FUNCTION_BLOCK logiBUS_QDA_PWM (* Composite FB for 13-bit PWM output data (0..8191 in DWORD) *)
  (* Standard: 61499-2; Description: Copyright (c) 2026 HR Agrartechnik GmbH This program and the accompanying materials are made available under the terms of the Eclipse Public License 2.0 which is available at https://www.eclipse.org/legal/epl-2.0/ SPDX-License-Identifier: EPL-2.0 *)
  (* Version 1.1, 2026-09-20, Franz Höpfinger, Meisterschulen am Ostbahnhof, Document 13-bit resolution (0..8191, 0..100% duty cycle) for OUT adapter socket *)
  (* Version 1.0, 2026-02-23, Franz Höpfinger, HR Agrartechnik GmbH *)
  PACKAGE logiBUS::io::DQ;
  IMPORT logiBUS::io::DQ::logiBUS_DO::Invalid;
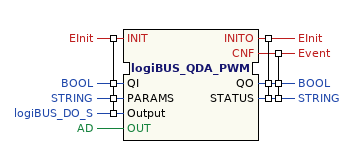
  EVENT_INPUT
    INIT : EInit WITH QI, PARAMS, Output; (* Service Initialization *)
  END_EVENT
  EVENT_OUTPUT
    INITO : EInit WITH QO, STATUS; (* Initialization Confirm *)
    CNF WITH QO, STATUS; (* Confirmation of Requested Service *)
  END_EVENT
  VAR_INPUT
    QI : BOOL; (* Event Input Qualifier *)
    PARAMS : STRING; (* Service Parameters *)
    Output : logiBUS::io::DQ::logiBUS_DO_S := Invalid; (* Identify the Output Output_Q1..Q8 *)
  END_VAR
  VAR_OUTPUT
    QO : BOOL; (* Event Output Qualifier *)
    STATUS : STRING; (* Service Status *)
  END_VAR
  SOCKETS
    OUT : adapter::types::unidirectional::AD; (* 13-bit raw PWM output data (0..8191, D1) *)
  END_SOCKETS
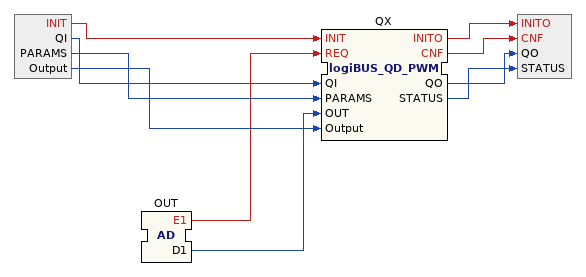
  FBS
    QX : logiBUS::io::DQ::logiBUS_QD_PWM;
  END_FBS
  EVENT_CONNECTIONS
    INIT TO QX.INIT;
    QX.INITO TO INITO;
    OUT.E1 TO QX.REQ;
    QX.CNF TO CNF;
  END_CONNECTIONS
  DATA_CONNECTIONS
    OUT.D1 TO QX.OUT;
    QI TO QX.QI;
    PARAMS TO QX.PARAMS;
    QX.QO TO QO;
    QX.STATUS TO STATUS;
    Output TO QX.Output;
  END_CONNECTIONS
END_FUNCTION_BLOCK
